TYPE (* CONSTANTS_MATH *)
  (* Description: ( * revision history hm	26.10.2008	rev 1.0 original version hm	26. mar. 2011	rev 1.1 added array facts * ) *)
  (* Version 1.0, 2025-12-21, Franz Höpfinger, initial API and implementation and/or initial documentation *)
  PACKAGE OSCAT::Basic::Data_types;
  CONSTANTS_MATH : STRUCT
    PI : REAL := 3.14159265358979323846264338327950288; (* Kreiszahl PI *)
    PI2 : REAL := 6.28318530717958647692528676655900576; (* PI * 2 *)
    PI4 : REAL := 12.56637061435917295385057353311801152; (* PI * 4 *)
    PI05 : REAL := 1.5707963267949; (* PI / 2 *)
    PI025 : REAL := 0.785398163397448; (* PI / 4 *)
    PI_INV : REAL := 0.318309886183791; (* 1 / PI *)
    EUL : REAL := 2.71828182845904523536028747135266249; (* Euler constant e *)
    E_INV : REAL := 0.367879441171442; (* 1 / e *)
    SQ2 : REAL := 1.4142135623731; (* Wurzel von 2 *)
    FACTS : ARRAY [0..12] OF DINT := [1,1,2,6,24,120,720,5040,40320,362880,3628800,39916800,479001600]; (* Factorials Array 0..12 *)
  END_STRUCT;
END_TYPE
